FUNCTION F_ForwardPropagation : LREAL
VAR_INPUT
	layer_pre : Layer;
	layer_next : Layer;
	pointer_in : POINTER TO LREAL;
	pointer_out : POINTER TO LREAL; 
END_VAR
VAR
	i : UINT;
	length_in : UINT;	
	length_out : UINT;

	activation_type : UINT;
END_VAR

length_in := layer_pre.num_neurons;
length_out := layer_next.num_neurons;
activation_type := layer_next.activation;
FOR i := 0 TO length_out-1 DO
	pointer_out[i] := F_Dot(ADR(layer_next.pointer_weight[i * length_in]),pointer_in,length_in); 
	pointer_out[i] := layer_next.pointer_bias[i] + pointer_out[i];
	CASE activation_type OF
		1:
		pointer_out[i] := F_relu(pointer_out[i]);
		2:
		pointer_out[i] := F_tanh(pointer_out[i]);
	ELSE
		CONTINUE;
	END_CASE
END_FOR

END_FUNCTION

(* stored: Version 1.1.0.1, ProductVersion 3.1.4024.12
   POU F_ForwardPropagation: Id {a4be79c7-1e65-45e2-ab2b-57c3b0f48949}, SpecialFunc None *)
